INTERFACE I_Position EXTENDS I_PosMover

PROPERTY RequestedStep : INT
GET
END_GET
SET
END_SET
END_PROPERTY

PROPERTY RequestMover : BOOL
GET
END_GET
END_PROPERTY

METHOD SetMoverLink : BOOL
VAR_INPUT
	mover : I_MoverPos;
END_VAR
END_METHOD

END_INTERFACE

(* stored: Version 1.1.0.1
   Itf I_Position: Id {48028eb2-2200-4fd3-b53c-8707e9a24ba1}
   Property RequestedStep: Id {04ed390e-b31b-40d6-ac18-4f6ca9de7e32}
   Get Get: Id {68767cb3-ce14-467d-afa2-dbd567bec1c2}
   Set Set: Id {e3481b16-81b9-4d39-ae75-5a5085a81a3f}
   Property RequestMover: Id {8cca03cd-3d79-4580-9113-4bd18f29085d}
   Get Get: Id {a22bf258-670e-4250-85e1-189b0613277c}
   Method SetMoverLink: Id {60187c0b-bede-4b3c-a1f4-276f700080c7} *)
